// TIA Portal V20 export
DATA_BLOCK "Parameter_Control"   // DB2
{ S7_Optimized_Access := 'TRUE' }
// stored: MemoryReserve 100
   VAR
      Sugar : Real;
      Salt : Int;
      Water : Int;
      Coffee_Powder : Int;
   END_VAR
BEGIN
END_DATA_BLOCK
